	IF iCountRemote>=20 THEN //累计20s认为时间可用
		iCountRemote:=20;
		dDelRTime := TO_ULINT(stUTC_Timestamp) - (dRTime + 8 * 3600 *1000);
		GVL.bRemoteTimeLock:=TRUE;
		//对外部和本机时间差做1分钟的均值滤波
	END_IF
	//GVL.dRemoteTime:=stUTC_Timestamp*1000000 - dMeanDelRTime;
	dLastRTime:=dRTime;
	(*
	IF GVL.bRemoteTimeLock THEN
		dCountRemote:= dCountRemote + 1;
		IF dCountRemote < 10000 THEN
			dMeanDelRTime := (dMeanDelRTime*(dCountRemote-1) + dDelRTime)/dCountRemote;
		ELSE
			dCountRemote := 10000;
			dMeanDelRTime := (dMeanDelRTime*(dCountRemote-1) + dDelRTime)/dCountRemote; 	
			//iDiff:=ULINT_TO_DINT(Gvl.dPTPCSTTime-dLastCSTtime);
			//dLastCSTtime:=dCSTTime;
		END_IF
	END_IF
	*)
END_IF

ulACUTimeStamp := stUTC_Timestamp - dDelRTime;

END_PROGRAM

// Device/Application/GPRMC_1_1
PROGRAM GPRMC_1_1
VAR
        com_init:gcan.FB_Com_Init;                      //gcan.FB_Com_Init为串口初始化功能块，可设定串口端口号，串口波特率等参数
        com_read:gcan.FB_Com_Read ;                                //gcan.FB_Com_Read为串口接收功能块，用于通过接收串口发送给PLC的数据
        com_write:gcan.FB_Com_Write ;                        //gcan.FB_Com_Write为串口发送功能块，用于发送串口数据
        m_uiError:UINT;                                                        //用于承接功能块中报错引脚错误信息的变量
        m_out:BOOL;                                                                //用于承接功能块中完成标志引脚数据的变量
        isFirst:BOOL:=TRUE;                                                //用于判断初始化只执行一次的逻辑
        mPort:BYTE;                                                                //程序中用作设定串口端口号
        recSize:UINT;                                                        //接收数据长度，单位：字节
        recBuf:ARRAY[0..120] OF BYTE;                        //用于存放接收到的串口数据的数组
        iYear: INT;                             //年
        iMonth: INT;                            //月
        iDay: INT;                              //日
        iHour: INT;                             //时
        iMinute: INT;                           //分
        iSecond: INT;                           //秒
    bChecksumValid: BOOL := FALSE;                //校验和
        nFrameHeadPos: INT := 0;                //帧头索引          
    nPos        : INT;                      //帧头位置
    nChecksumRx : BYTE := 0;                //和校验
        strDateTimeNow : STRING;
        gnssTimestamp: ULINT;
        gnssTimestamplast:ULINT;
        icount:INT;
END_VAR

////////////////////////////////////////////////////////////////////////////////////////
//串口接收TOD报文解析
//日期：2025/05/15
//版本：V1.1
/////////////////////////////////////////////////////////////////////////////////////////

mPort:=1;                                                                //串口端口号设定，GCAN-PLC-400、GCAN-PLC-510、GCAN-PLC-511，1为232，2为485
                                                                                //GCAN-PLC-324、GCAN-PLC-326，1为第一路485，2为第2路485
IF isFirst THEN
        com_init(                                                        //串口初始化功能块
        EN_IN:=TRUE,                                                //串口初始化功能块使能
        xEnable:=TRUE,                                                //串口功能使能
        bPort:=mPort,                                                //串口端口号设定
        uiBaudrate:=115200,                                        //串口波特率设定
        bParity:=0,                                                        //串口奇偶校验设定，0为无校验，1为奇校验，2为偶检验
        bDatabits:=8,                                                //数据位设定
        bStopbits:=1,                                                //停止位设定
        EN_OUT=>m_out,                                                //串口初始化功能块执行完成标志位
        uiError=>m_uiError);                                //串口初始化功能块执行错误信息
        isfirst:=FALSE;                                                //执行一次初始化后关闭IF的条件使其之后进入ELSE程序段运行

ELSE
        
                com_read(                                                //串口读取功能块
                EN_in:=TRUE,                                        //读取功能块使能，为TRUE执行读取
                bPort:=mPort,                                        //串口端口号设定
                p_brxdata:=ADR(recBuf),                        //读取到的串口数据引脚为指针类型，使用ADR()指向自建数组将数据存放到数组中
                uiMaxsize:=240,                                        //设定最大读取长度
                EN_out=>m_out,                                        //串口读取功能块执行完成标志位******功能块执行完成不代表接收完成********
                uiRecSize=>recSize,                                //串口接收数据长度，单位：字节，大于0时说明接收到数据可用于判断是否接收
                uierror=>m_uierror);                        //串口读取功能块执行错误信息
                // 查找帧头 $X (36, 88)
                FOR nPos := 0 TO 119 DO
                        IF recBuf[nPos] = 36 AND recBuf[nPos + 1] = 88 THEN
                                nFrameHeadPos := nPos;
                                EXIT;
                        END_IF
                END_FOR
                //解析时间日期 
                IF nFrameHeadPos + 26 <= 120 THEN
                        iYear:=BYTE_TO_INT(recBuf[nFrameHeadPos+23]-48)*1000+BYTE_TO_INT(recBuf[nFrameHeadPos+24]-48)*100+BYTE_TO_INT(recBuf[nFrameHeadPos+25]-48)*10+BYTE_TO_INT(recBuf[26]-48);
                        iMonth:=BYTE_TO_INT(recBuf[nFrameHeadPos+20]-48)*10+BYTE_TO_INT(recBuf[nFrameHeadPos+21]-48);
                        iDay:=BYTE_TO_INT(recBuf[nFrameHeadPos+17]-48)*10+BYTE_TO_INT(recBuf[nFrameHeadPos+18]-48);
                        iHour:=BYTE_TO_INT(recBuf[nFrameHeadPos+7]-48)*10+BYTE_TO_INT(recBuf[nFrameHeadPos+8]-48)+8;
                        iMinute:=BYTE_TO_INT(recBuf[nFrameHeadPos+9]-48)*10+BYTE_TO_INT(recBuf[nFrameHeadPos+10]-48);
                        iSecond:=BYTE_TO_INT(recBuf[nFrameHeadPos+11]-48)*10+BYTE_TO_INT(recBuf[nFrameHeadPos+12]-48);
                        // 计算时间戳                
                        
                        strDateTimeNow := CONCAT(STR1 := 'DT#', STR2 := INT_TO_STRING(iYear));
                        strDateTimeNow := CONCAT(STR1 := strDateTimeNow, STR2 := '-');
                        strDateTimeNow := CONCAT(STR1 := strDateTimeNow, STR2 := INT_TO_STRING(iMonth));
                        strDateTimeNow := CONCAT(STR1 := strDateTimeNow, STR2 := '-');
                        strDateTimeNow := CONCAT(STR1 := strDateTimeNow, STR2 := INT_TO_STRING(iDay));
                        strDateTimeNow := CONCAT(STR1 := strDateTimeNow, STR2 := '-');
                        strDateTimeNow := CONCAT(STR1 := strDateTimeNow, STR2 := INT_TO_STRING(iHour));
                        strDateTimeNow := CONCAT(STR1 := strDateTimeNow, STR2 := ':');
                        strDateTimeNow := CONCAT(STR1 := strDateTimeNow, STR2 := INT_TO_STRING(iMinute));
                        strDateTimeNow := CONCAT(STR1 := strDateTimeNow, STR2 := ':');
                        strDateTimeNow := CONCAT(STR1 := strDateTimeNow, STR2 := INT_TO_STRING(iSecond));
                        
                        gnssTimestamplast:=gnssTimestamp;
                        gnssTimestamp := DT_TO_ULINT(TO_DT(strDateTimeNow)) * 1000;
                        GVL.stGNSS_Timestap := gnssTimestamp;                        
                END_IF
                
                IF gnssTimestamplast<>gnssTimestamp THEN
                        icount:=0;
                ELSE
                        icount:=icount+1;
                END_IF        
END_IF

END_PROGRAM

// Device/Application/PID_1
FUNCTION_BLOCK PID_1
VAR_INPUT
    rTarget : REAL;       (* 设定值 *)
    rFeedback : REAL;       (* 反馈值 *)
	rPosLimPositive:LREAL;//位置正限位
	rPosLimNegative:LREAL;//位置反限位
	rKp:REAL;     //比例增益
	rKi:REAL;     //积分增益
	rKd:REAL;     //微分增益
	iThreshold:INT;//积分项开启的位置阈值
	bPIDEnable:BOOL:=TRUE;//PID使能
	rVelLim:LREAL;//速度限制
END_VAR
VAR_OUTPUT
    rPIDOutput : LREAL:=0;         //带方向的输出速度

END_VAR
VAR
	//rPIDOutPut: REAL:=0.0;
	rLastError: LREAL:=0.0;(*上一次误差*)
	rErrorNow:LREAL:=0.0;(*当前误差*)
    rIntegralNew : LREAL := 0.0; (* 积分项 *)
    rDerivativeNew : LREAL := 0.0; (* 微分项 *)
	rDelta: LREAL;(*增量*)
	rProportionNew: LREAL;
	
	//iAzPIDEnable: INT;
END_VAR


IF (bPIDEnable>0) THEN //如果PID使能
	IF rTarget=rFeedback THEN
		rPIDOutput:=0;	
	ELSE
	
		rErrorNow:=rTarget-rFeedback;//计算当前误差 en
		rProportionNew:=rErrorNow;//比例项
		//积分项
		IF rFeedback>rPosLimNegative AND rFeedback<rPosLimPositive THEN //若在软限位之内，工作时开启积分项
			IF (ABS(rTarget-rFeedback)<iThreshold OR iThreshold = -1) THEN//位置差小于积分阈值开始积分，或者设置阈值为-1，不启用这个控制
				rIntegralNew:= rIntegralNew+rErrorNow; //积分项
			ELSE
				rIntegralNew:=0;
			END_IF;
		ELSE //不在软限位范围内,则积分项为0
			rIntegralNew:=0;
		END_IF

		//PID输出
		rPIDOutPut:=rKp*rProportionNew+rKi*rIntegralNew;


		//PID限速
		
			IF rPIDOutput<(-rVelLim) THEN
				rPIDOutput:=-rVelLim;
			ELSIF rPIDOutput>rVelLim THEN
				rPIDOutput:=rVelLim;
			END_IF
		
		
		IF rFeedback>rPosLimPositive AND rPIDOutput>0 THEN 
			rPIDOutput:=0;
		END_IF
		IF rFeedback<rPosLimNegative AND rPIDOutput<0 THEN
			rPIDOutput:=0;
		END_IF
		
		rLastError:=rErrorNow;//将当前误差赋值给上一次误差
		
	END_IF
ELSE//非使能清零PID各项
	rProportionNew:=0.0;
	rIntegralNew:=0.0;
	rPIDOutput:=0.0;
END_IF

END_FUNCTION_BLOCK

// Device/Application/PLC_PRG
PROGRAM PLC_PRG
VAR
	a : DINT;
	b : REAL;
END_VAR

a := REAL_TO_DINT(b * 524288 / 360);

END_PROGRAM

// Device/Application/XPTOD_SerialCom
PROGRAM XPTOD_SerialCom
VAR
        com_init:gcan.FB_Com_Init;                      //gcan.FB_Com_Init为串口初始化功能块，可设定串口端口号，串口波特率等参数
        com_read:gcan.FB_Com_Read ;                                //gcan.FB_Com_Read为串口接收功能块，用于通过接收串口发送给PLC的数据
        com_write:gcan.FB_Com_Write ;                        //gcan.FB_Com_Write为串口发送功能块，用于发送串口数据
        m_uiError:UINT;                                                        //用于承接功能块中报错引脚错误信息的变量
        m_out:BOOL;                                                                //用于承接功能块中完成标志引脚数据的变量
        isFirst:BOOL:=TRUE;                                                //用于判断初始化只执行一次的逻辑
        mPort:BYTE;                                                                //程序中用作设定串口端口号
        recSize:UINT;                                                        //接收数据长度，单位：字节
        recBuf:ARRAY[0..239] OF BYTE;                        //用于存放接收到的串口数据的数组
        iYear: INT;                             //年
        iMonth: INT;                            //月
        iDay: INT;                              //日
        iHour: INT;                             //时
        iMinute: INT;                           //分
        iSecond: INT;                           //秒
    bChecksumValid: BOOL := FALSE;                //校验和
        nFrameHeadPos: INT := 0;                //帧头索引          
    nPos        : INT;                      //帧头位置
    nChecksumRx : BYTE := 0;                //和校验
        strDateTimeNow : STRING;
        gnssTimestamp: ULINT;
        gnssTimestamplast:ULINT;
        icount:INT;
END_VAR

////////////////////////////////////////////////////////////////////////////////////////
//串口接收TOD报文解析
//日期：2025/05/15
//版本：V1.1
/////////////////////////////////////////////////////////////////////////////////////////

mPort:=1;                                                                //串口端口号设定，GCAN-PLC-400、GCAN-PLC-510、GCAN-PLC-511，1为232，2为485
                                                                                //GCAN-PLC-324、GCAN-PLC-326，1为第一路485，2为第2路485
IF isFirst THEN
        com_init(                                                        //串口初始化功能块
        EN_IN:=TRUE,                                                //串口初始化功能块使能
        xEnable:=TRUE,                                                //串口功能使能
        bPort:=mPort,                                                //串口端口号设定
        uiBaudrate:=115200,                                        //串口波特率设定
        bParity:=0,                                                        //串口奇偶校验设定，0为无校验，1为奇校验，2为偶检验
        bDatabits:=8,                                                //数据位设定
        bStopbits:=1,                                                //停止位设定
        EN_OUT=>m_out,                                                //串口初始化功能块执行完成标志位
        uiError=>m_uiError);                                //串口初始化功能块执行错误信息
        isfirst:=FALSE;                                                //执行一次初始化后关闭IF的条件使其之后进入ELSE程序段运行

ELSE
        
                com_read(                                                //串口读取功能块
                EN_in:=TRUE,                                        //读取功能块使能，为TRUE执行读取
                bPort:=mPort,                                        //串口端口号设定
                p_brxdata:=ADR(recBuf),                        //读取到的串口数据引脚为指针类型，使用ADR()指向自建数组将数据存放到数组中
                uiMaxsize:=240,                                        //设定最大读取长度
                EN_out=>m_out,                                        //串口读取功能块执行完成标志位******功能块执行完成不代表接收完成********
                uiRecSize=>recSize,                                //串口接收数据长度，单位：字节，大于0时说明接收到数据可用于判断是否接收
                uierror=>m_uierror);                        //串口读取功能块执行错误信息
                // 查找帧头 $X (36, 88)
                FOR nPos := 1 TO 240 DO
                        IF recBuf[nPos] = 36 AND recBuf[nPos + 1] = 88 THEN
                                nFrameHeadPos := nPos;
                                EXIT;
                        END_IF
                END_FOR
                //解析时间日期 
                IF nFrameHeadPos + 26 <= 240 THEN
                        iYear:=BYTE_TO_INT(recBuf[nFrameHeadPos+23]-48)*1000+BYTE_TO_INT(recBuf[nFrameHeadPos+24]-48)*100+BYTE_TO_INT(recBuf[nFrameHeadPos+25]-48)*10+BYTE_TO_INT(recBuf[26]-48);
                        iMonth:=BYTE_TO_INT(recBuf[nFrameHeadPos+20]-48)*10+BYTE_TO_INT(recBuf[nFrameHeadPos+21]-48);
                        iDay:=BYTE_TO_INT(recBuf[nFrameHeadPos+17]-48)*10+BYTE_TO_INT(recBuf[nFrameHeadPos+18]-48);
                        iHour:=BYTE_TO_INT(recBuf[nFrameHeadPos+7]-48)*10+BYTE_TO_INT(recBuf[nFrameHeadPos+8]-48)+8;
                        iMinute:=BYTE_TO_INT(recBuf[nFrameHeadPos+9]-48)*10+BYTE_TO_INT(recBuf[nFrameHeadPos+10]-48);
                        iSecond:=BYTE_TO_INT(recBuf[nFrameHeadPos+11]-48)*10+BYTE_TO_INT(recBuf[nFrameHeadPos+12]-48);
                        // 计算时间戳                
                        
                        strDateTimeNow := CONCAT(STR1 := 'DT#', STR2 := INT_TO_STRING(iYear));
                        strDateTimeNow := CONCAT(STR1 := strDateTimeNow, STR2 := '-');
                        strDateTimeNow := CONCAT(STR1 := strDateTimeNow, STR2 := INT_TO_STRING(iMonth));
                        strDateTimeNow := CONCAT(STR1 := strDateTimeNow, STR2 := '-');
                        strDateTimeNow := CONCAT(STR1 := strDateTimeNow, STR2 := INT_TO_STRING(iDay));
                        strDateTimeNow := CONCAT(STR1 := strDateTimeNow, STR2 := '-');
                        strDateTimeNow := CONCAT(STR1 := strDateTimeNow, STR2 := INT_TO_STRING(iHour));
                        strDateTimeNow := CONCAT(STR1 := strDateTimeNow, STR2 := ':');
                        strDateTimeNow := CONCAT(STR1 := strDateTimeNow, STR2 := INT_TO_STRING(iMinute));
                        strDateTimeNow := CONCAT(STR1 := strDateTimeNow, STR2 := ':');
                        strDateTimeNow := CONCAT(STR1 := strDateTimeNow, STR2 := INT_TO_STRING(iSecond));
                        
                        gnssTimestamplast:=gnssTimestamp;
                        gnssTimestamp := DT_TO_ULINT(TO_DT(strDateTimeNow)) * 1000;
                        GVL.stGNSS_Timestap := gnssTimestamp;                        
                END_IF
                
                IF gnssTimestamplast<>gnssTimestamp THEN
                        icount:=0;
                ELSE
                        icount:=icount+1;
                END_IF        
END_IF

END_PROGRAM

// Device/Application/插值模块/InterDataProcess
FUNCTION_BLOCK InterDataProcess
VAR_INPUT
	ulRealTime: ULINT;//实际时间 单位纳秒
	//aOrbitTime: ARRAY [1..5] OF ULINT;//轨道时间数组
	Arr: ARRAY [1..5] OF ULINT:=[9,0,1,5,4]; // 创建一个包含5个整数的数组 轨道时间数组  起点 1970-01-01 0:00:00 单位纳秒
    
END_VAR
VAR_OUTPUT
	MaxVal, MinVal: ULINT;   // 定义最大值、最小值和循环计数器变量
    MaxIndex, MinIndex: INT; // 定义最大值和最小值的索引
	ulInterRealTime : ULINT;//插值使用的时间
END_VAR
VAR
	i,j: INT;
END_VAR

//该功能块查找到轨道时间数组内最大最小值以及索引位置
//找出最大最小值
MaxVal := 0; // 初始化最大值
MinVal := 0; // 初始化最小值
MaxIndex := 0; // 初始化最大值的索引
MinIndex := 0; // 初始化最小值的索引

FOR i := 1 TO 5 DO
    IF Arr[i] <> 0 THEN
        IF MaxVal = 0 THEN
            MaxVal := Arr[i];
            MaxIndex := i;
        ELSIF Arr[i] > MaxVal THEN
            MaxVal := Arr[i];
            MaxIndex := i;
        END_IF

        IF MinVal = 0 THEN
            MinVal := Arr[i];
            MinIndex := i;
        ELSIF Arr[i] < MinVal THEN
            MinVal := Arr[i];
            MinIndex := i;
        END_IF
    END_IF
END_FOR

// MaxVal 和 MinVal 包含了最大值和最小值，不考虑值为0的元素
// MaxIndex 和 MinIndex 包含了最大值和最小值的索引


//当前时间和最大最小比较 
IF ulRealTime<MinVal*1000000 THEN //小于插值范围 取最小时间
	//
	ulInterRealTime:=MinVal*1000000; //应该修改插值位置 而不是时间
ELSIF ulRealTime>MaxVal*1000000THEN //大于插值范围 取最大时间
	//
	ulInterRealTime:=MaxVal*1000000;//应该修改插值位置 而不是时间
ELSE
	//如果内部有0 则不插值选取最新的数据
	FOR j:=1 TO 5 DO
		IF (Arr[i]=0) AND (j<5) THEN
			ulInterRealTime:=Arr[5];//应该修改插值位置 而不是时间
			MaxIndex:=5;
			EXIT;
		ELSIF (Arr[i]=0) AND (j=5) THEN
			//没有输入数据 需要报错吗？
		END_IF
	END_FOR
	//
END_IF

END_FUNCTION_BLOCK

// Device/Application/插值模块/LinearInter
FUNCTION_BLOCK LinearInter
VAR_INPUT
	tLastTime:ULINT;//上一时间
	rLastPos:REAL;//上一时间位置
	
	tCurTime:ULINT;//当前时间
	rCurPos:REAL;//当前时间位置
	
	tTargetTime:ULINT;//目标时间
END_VAR
VAR_OUTPUT
	rTargetpos:REAL;//目标时间位置
END_VAR
VAR
	iDelCurLastTime:LREAL:=1.0;//	当前与上一个时间差
	iDelTarCurTime:LREAL:=1.0;//目标与当前时间差
	rK:REAL;//方位斜率
END_VAR

//tLastTime:=tLastTime/1000000;
//tCurTime:=tCurTime/1000000;
//tTargetTime:=tTargetTime/1000000;
iDelTarCurTime:=ULINT_TO_LREAL(tTargetTime)-ULINT_TO_LREAL(tCurTime); //x1-x
IF (tCurTime-tLastTime)<>0 THEN
	iDelCurLastTime:=ULINT_TO_LREAL(tCurTime)-ULINT_TO_LREAL(tLastTime);  //x-x0
ELSE
	iDelCurLastTime:=1.0;
END_IF

IF iDelTarCurTime<>0 THEN
	rK:=(rCurPos-rLastPos)/(iDelCurLastTime);
ELSE
	rK:=0;
END_IF
rTargetpos:=rCurPos+rK*iDelTarCurTime;  //y1 + ((y1-y0)/(x1-x0))*(x-x1)

END_FUNCTION_BLOCK

// Device/Application/插值模块/threesimple2
FUNCTION_BLOCK threesimple2
VAR_INPUT
	aUTC_TIME:ARRAY [1..5] OF ULINT;  //用于三次样条插值的数据
	aPosCmd :ARRAY [1..5] OF LREAL;//用于三次样条插值的数据
	
	y0:REAL;
	yn:REAL;//y0,yn表示的是S''(x0)=f''(x0)=y0，S''(xn)=f''(xn)=yn,自然边界即条件值为0
	xt:REAL;//所求目标位置
END_VAR
VAR_OUTPUT
	sout:REAL;
	nout:INT;
END_VAR
VAR
	Three:three2;
	X:ARRAY [1..5] OF LREAL;
	Y:ARRAY [1..5] OF LREAL;
	M :ARRAY [1..5] OF LREAL;
	A: ARRAY [1..5,1..5] OF LREAL;
	D: ARRAY[1..3,1..3] OF LREAL;
	g: ARRAY [1..3] OF LREAL;
	h:ARRAY [1..4] OF LREAL;
	
	n:INT:=5;
	
	p1: ARRAY [1..4] OF REAL;
	p2:ARRAY [1..4] OF REAL;
	p3:ARRAY [1..4] OF REAL;
	p4:ARRAY [1..4] OF REAL;
	i:INT;
	
END_VAR

FOR i:=1 TO 5 DO
	X[i]:=ULINT_TO_LREAL(aUTC_TIME[i]);
	Y[i]:=aPosCmd[i];
END_FOR


Three(X:=X,Y:=Y,y0:=y0,yn:=yn,D=>D,h=>h,A=>A,g=>g,M=>M);

FOR i:=1 TO (n-1) DO
	p1[i]:=M[i]*(X[i+1]-xt)*(X[i+1]-xt)*(X[i+1]-xt)/(6*h[i]);
	p2[i]:=M[i+1]*(xt-X[i])*(xt-X[i])*(xt-X[i])/(6*h[i]);
	p3[i]:=(A[i,1]-M[i]/6*(h[i])*(h[i]))*(X[i+1]-xt)/h[i];
	p4[i]:=(A[i+1,1]-M[i+1]/6*(h[i])*(h[i]))*(xt-X[i])/h[i];
	
	
END_FOR


FOR i:=1 TO (n-1) DO
	IF (xt<=X[i+1])AND (xt>=X[i]) THEN
		nout:=i;
		sout:=p1[nout]+p2[nout]+p3[nout]+p4[nout]; 
	ELSIF xt>X[5] THEN
		nout:=4;
	ELSIF xt<X[1]THEN
		nout:=1;
	END_IF
END_FOR


//要不要判断插值模块是否有效？
sout:=p1[nout]+p2[nout]+p3[nout]+p4[nout]; 
(*
IF xt>X[5] THEN
	nout:=4;
	sout:=p1[nout]+p2[nout]+p3[nout]+p4[nout]; 
ELSIF xt<X[1] THEN
	nout:=1;
	sout:=p1[nout]+p2[nout]+p3[nout]+p4[nout]; 
END_IF
*)

END_FUNCTION_BLOCK

// /ElCtrl
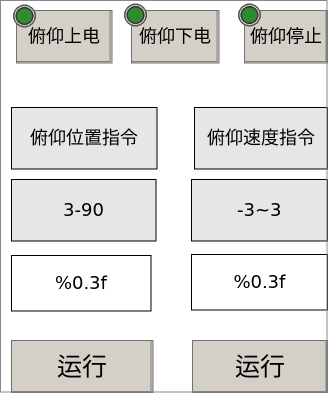
VISUALIZATION ElCtrl  // 328x393
    Button (131,10 88x53), "俯仰下电"
        OnMouseClick: execute { GVL.Axis1Local.iMode:=0; }
    Button (16,10 96x53), "俯仰上电"
        OnMouseClick: execute { GVL.Axis1Local.iMode:=1; }
    Lamp1 (6,3 37x26), variable: GVL.Axis1Status.bServo_Enable, style: Lamp-Lamp1-Green
    Lamp1 (117,2 37x26), variable: NOT(GVL.Axis1Status.bServo_Enable), style: Lamp-Lamp1-Green
    Button (244,10 84x53), "俯仰停止"
        OnMouseClick: execute { GVL.Axis1Local.iMode:=7; }
    Lamp1 (231,2 37x26), variable: NOT(GVL.Axis1Status.Moving), style: Lamp-Lamp1-Green
    Rectangle (11,107 146x62), "俯仰位置指令"
    Rectangle (11,255 140x56), "%0.3f", text variable: ElV.rPosCmd
        OnMouseClick: write the text variable via Default, min 3, max 90
    Button (11,340 142x53), "运行"
        OnMouseClick: execute {
            GVL.Axis1Local.rPosCmd:=GVL.ElV.rPosCmd+90;
            GVL.Axis1Local.iMode:=4;
            GVL.Axis1Local.bPIDEnable:=TRUE;
        }
    Rectangle (194,107 134x62), "俯仰速度指令"
    Rectangle (191,254 137x56), "%0.3f", text variable: ElV.rVelCmd
        OnMouseClick: write the text variable via Default, min -10, max 10
    Button (192,340 136x53), "运行"
        OnMouseClick: execute { GVL.Axis1Local.rVelCmd:=GVL.ElV.rVelCmd; GVL.Axis1Local.iMode:=3; }
    Rectangle (11,179 145x62), "3-90"
    Rectangle (191,179 137x62), "-3~3"
END_VISUALIZATION

// Device/Application/可视化/AzCtrl
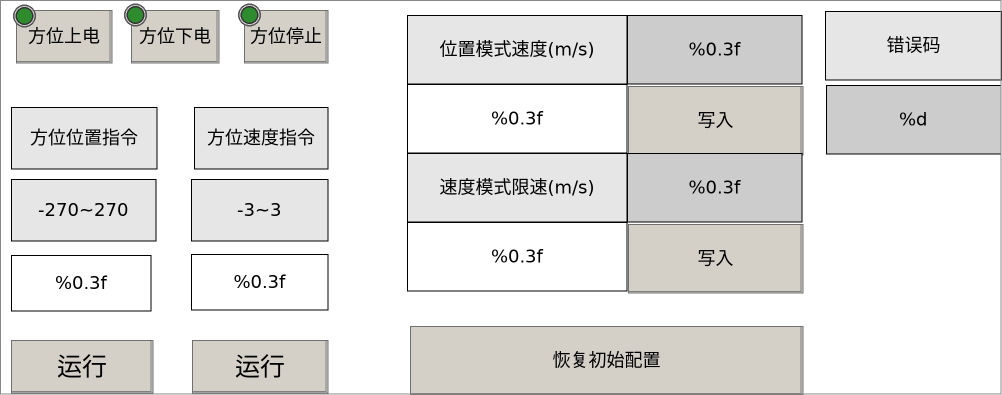
VISUALIZATION AzCtrl  // 1002x395
    Button (131,10 88x53), "方位下电"
        OnMouseClick: execute { GVL.Axis2Local.iMode:=0; }
    Button (16,10 96x53), "方位上电"
        OnMouseClick: execute { GVL.Axis2Local.iMode:=1; }
    Lamp1 (6,3 37x26), variable: GVL.Axis2Status.bServo_Enable, style: Lamp-Lamp1-Green
    Lamp1 (117,2 37x26), variable: NOT(GVL.Axis2Status.bServo_Enable), style: Lamp-Lamp1-Green
    Button (244,10 84x53), "方位停止"
        OnMouseClick: execute { GVL.Axis2Local.iMode:=7; }
    Lamp1 (231,2 37x26), variable: NOT(GVL.Axis2Status.Moving), style: Lamp-Lamp1-Green
    Rectangle (11,107 146x62), "方位位置指令"
    Rectangle (11,255 140x56), "%0.3f", text variable: AzV.rPosCmd
        OnMouseClick: write the text variable via Default, min -270, max 270
    Button (11,340 142x53), "运行"
        OnMouseClick: execute {
            GVL.Axis2Local.rPosCmd:=-GVL.AzV.rPosCmd;
            GVL.Axis2Local.iMode:=4;
            GVL.Axis2Local.bPIDEnable:=TRUE;
        }
    Rectangle (194,107 134x62), "方位速度指令"
    Rectangle (191,254 137x56), "%0.3f", text variable: AzV.rVelCmd
        OnMouseClick: write the text variable via Default, min -20, max 20
    Button (192,340 136x53), "运行"
        OnMouseClick: execute { GVL.Axis2Local.rVelCmd:=GVL.AzV.rVelCmd*(-1); GVL.Axis2Local.iMode:=3; }
    Rectangle (11,179 145x62), "-270~270"
    Rectangle (191,179 137x62), "-3~3"
    Rectangle (627,15 175x69), "%0.3f", text variable: Axis2Local.Pos_Vel
    Rectangle (407,15 220x69), "位置模式速度(m/s)"
    Rectangle (407,84 220x69), "%0.3f", text variable: AzV.Pos_Vel
        OnMouseClick: write the text variable via Edit, min -15.5, max 15.5
    Button (628,86 175x69), "写入"
        OnMouseClick: execute { Axis2Local.Pos_Vel:=AzV.Pos_Vel; }
    Rectangle (627,153 175x69), "%0.3f", text variable: Axis2Local.rVel_Limit
    Rectangle (407,153 220x69), "速度模式限速(m/s)"
    Rectangle (407,222 220x69), "%0.3f", text variable: AzV.rVel_Limit
        OnMouseClick: write the text variable via Edit, min 2, max 15.5
    Button (628,224 175x69), "写入"
        OnMouseClick: execute { Axis2Local.rVel_Limit:=AzV.rVel_Limit; }
    Button (410,326 393x69), "恢复初始配置"
        OnMouseClick: execute { Axis2Local.rVel_Limit:=3; Axis2Local.Pos_Vel:=4; }
    Rectangle (826,85 175x69), "%d", text variable: GVL.eAzErrorcode
    Rectangle (825,11 177x69), "错误码"
END_VISUALIZATION

// Device/Application/可视化/ElCtrl
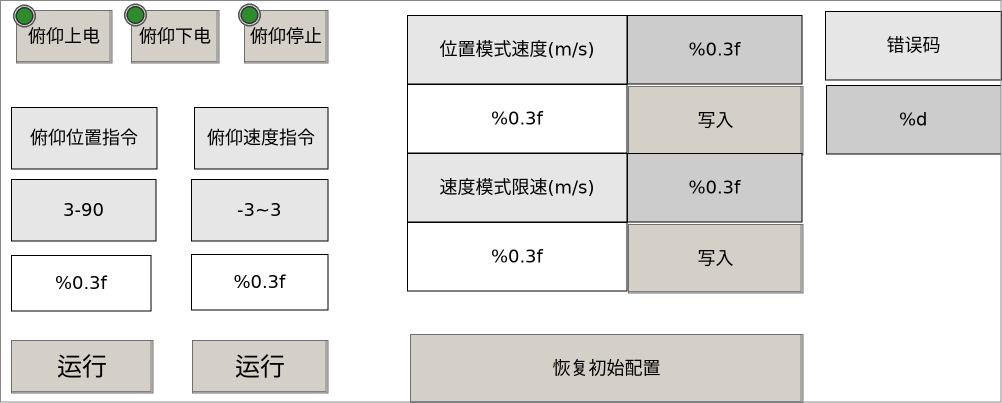
VISUALIZATION ElCtrl  // 1002x403
    Button (131,10 88x53), "俯仰下电"
        OnMouseClick: execute { GVL.Axis1Local.iMode:=0; }
    Button (16,10 96x53), "俯仰上电"
        OnMouseClick: execute { GVL.Axis1Local.iMode:=1; }
    Lamp1 (6,3 37x26), variable: GVL.Axis1Status.bServo_Enable, style: Lamp-Lamp1-Green
    Lamp1 (117,2 37x26), variable: NOT(GVL.Axis1Status.bServo_Enable), style: Lamp-Lamp1-Green
    Button (244,10 84x53), "俯仰停止"
        OnMouseClick: execute { GVL.Axis1Local.iMode:=7; }
    Lamp1 (231,2 37x26), variable: NOT(GVL.Axis1Status.Moving), style: Lamp-Lamp1-Green
    Rectangle (11,107 146x62), "俯仰位置指令"
    Rectangle (11,255 140x56), "%0.3f", text variable: ElV.rPosCmd
        OnMouseClick: write the text variable via Default, min 0, max 90
    Button (11,340 142x53), "运行"
        OnMouseClick: execute {
            GVL.Axis1Local.rPosCmd:=GVL.ElV.rPosCmd+90;
            GVL.Axis1Local.iMode:=4;
            GVL.Axis1Local.bPIDEnable:=TRUE;
        }
    Rectangle (194,107 134x62), "俯仰速度指令"
    Rectangle (191,254 137x56), "%0.3f", text variable: ElV.rVelCmd
        OnMouseClick: write the text variable via Default, min -13, max 13
    Button (192,340 136x53), "运行"
        OnMouseClick: execute { GVL.Axis1Local.rVelCmd:=GVL.ElV.rVelCmd; GVL.Axis1Local.iMode:=3; }
    Rectangle (11,179 145x62), "3-90"
    Rectangle (191,179 137x62), "-3~3"
    Rectangle (627,15 175x69), "%0.3f", text variable: Axis1Local.Pos_Vel
    Rectangle (407,15 220x69), "位置模式速度(m/s)"
    Rectangle (407,84 220x69), "%0.3f", text variable: ElV.Pos_Vel
        OnMouseClick: write the text variable via Edit, min -15.5, max 15.5
    Button (628,86 175x69), "写入"
        OnMouseClick: execute { Axis1Local.Pos_Vel:=ElV.Pos_Vel; }
    Rectangle (627,153 175x69), "%0.3f", text variable: Axis1Local.rVel_Limit
    Rectangle (407,153 220x69), "速度模式限速(m/s)"
    Rectangle (407,222 220x69), "%0.3f", text variable: ElV.rVel_Limit
        OnMouseClick: write the text variable via Edit, min 2, max 11
    Button (628,224 175x69), "写入"
        OnMouseClick: execute { Axis1Local.rVel_Limit:=ElV.rVel_Limit; }
    Button (410,334 393x69), "恢复初始配置"
        OnMouseClick: execute { Axis1Local.rVel_Limit:=3; Axis1Local.Pos_Vel:=4; }
    Rectangle (826,85 175x69), "%d", text variable: GVL.eElErrorcode
    Rectangle (825,11 177x69), "错误码"
END_VISUALIZATION

// Device/Application/可视化/north
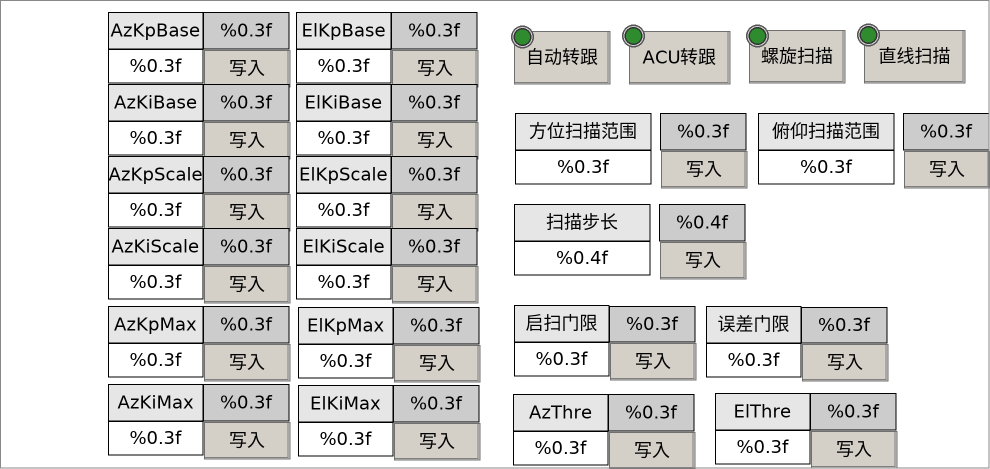
VISUALIZATION north  // 990x469
    Rectangle (203,12 86x37), "%0.3f", text variable: PersistentVars.rAzKpBase
    Rectangle (108,12 95x37), "AzKpBase"
    Rectangle (108,49 95x34), "%0.3f", text variable: GVL.rvAzKpBase
        OnMouseClick: write the text variable via Edit, min -100, max 100
    Button (204,50 86x37), "写入"
        OnMouseClick: execute { persistentvars.rAzKpBase := gvl.rvAzKpBase; }
    Rectangle (203,84 86x37), "%0.3f", text variable: PersistentVars.rAzKiBase
    Button (204,122 86x37), "写入"
        OnMouseClick: execute { persistentvars.rAzKiBase := gvl.rvAzKiBase; }
    Rectangle (203,156 86x37), "%0.3f", text variable: PersistentVars.rAzKpscale
    Button (204,194 86x37), "写入"
        OnMouseClick: execute { persistentvars.rAzKpScale := gvl.rvAzKpScale; }
    Rectangle (203,228 86x37), "%0.3f", text variable: PersistentVars.rAzKiscale
    Button (204,266 86x37), "写入"
        OnMouseClick: execute { persistentvars.rAzKiScale := gvl.rvAzKiScale; }
    Rectangle (108,84 95x37), "AzKiBase"
    Rectangle (108,121 95x34), "%0.3f", text variable: GVL.rvAzKiBase
        OnMouseClick: write the text variable via Edit, min -100, max 100
    Rectangle (108,156 95x37), "AzKpScale"
    Rectangle (108,193 95x34), "%0.3f", text variable: GVL.rvAzKpscale
        OnMouseClick: write the text variable via Edit, min -100, max 100
    Rectangle (108,228 95x37), "AzKiScale"
    Rectangle (108,265 95x34), "%0.3f", text variable: GVL.rvAzKiscale
        OnMouseClick: write the text variable via Edit, min -100, max 100
    Rectangle (391,12 86x37), "%0.3f", text variable: PersistentVars.rElKpBase
    Rectangle (296,12 95x37), "ElKpBase"
    Rectangle (296,49 95x34), "%0.3f", text variable: GVL.rvElKpBase
        OnMouseClick: write the text variable via Edit, min -100, max 100
    Button (392,50 86x37), "写入"
        OnMouseClick: execute { persistentvars.rElKpBase := gvl.rvElKpBase; }
    Rectangle (391,84 86x37), "%0.3f", text variable: PersistentVars.rElKiBase
    Button (392,122 86x37), "写入"
        OnMouseClick: execute { persistentvars.rElKiBase := gvl.rvElKiBase; }
    Rectangle (391,156 86x37), "%0.3f", text variable: PersistentVars.rElKpscale
    Button (392,194 86x37), "写入"
        OnMouseClick: execute { persistentvars.rElKpScale := gvl.rvElKpScale; }
    Rectangle (391,228 86x37), "%0.3f", text variable: PersistentVars.rElKiscale
    Button (392,266 86x37), "写入"
        OnMouseClick: execute { persistentvars.rElKiScale := gvl.rvElKiScale; }
    Rectangle (296,84 95x37), "ElKiBase"
    Rectangle (296,121 95x34), "%0.3f", text variable: GVL.rvElKiBase
        OnMouseClick: write the text variable via Edit, min -100, max 100
    Rectangle (296,156 95x37), "ElKpScale"
    Rectangle (296,193 95x34), "%0.3f", text variable: GVL.rvElKpscale
        OnMouseClick: write the text variable via Edit, min -100, max 100
    Rectangle (296,228 95x37), "ElKiScale"
    Rectangle (296,265 95x34), "%0.3f", text variable: GVL.rvElKiscale
        OnMouseClick: write the text variable via Edit, min -100, max 100
    Rectangle (203,306 86x37), "%0.3f", text variable: PersistentVars.rAzKpMax
    Rectangle (108,306 95x37), "AzKpMax"
    Rectangle (108,343 95x34), "%0.3f", text variable: GVL.rvAzKpMax
        OnMouseClick: write the text variable via Edit, min -100, max 100
    Button (204,344 86x37), "写入"
        OnMouseClick: execute { persistentvars.rAzKpMax := gvl.rvAzKpMax; }
    Rectangle (203,384 86x37), "%0.3f", text variable: PersistentVars.rAzKiMax
    Rectangle (108,384 95x37), "AzKiMax"
    Rectangle (108,421 95x34), "%0.3f", text variable: GVL.rvAzKiMax
        OnMouseClick: write the text variable via Edit, min -100, max 100
    Button (204,422 86x37), "写入"
        OnMouseClick: execute { persistentvars.rAzKiMax := gvl.rvAzKiMax; }
    Rectangle (393,307 86x37), "%0.3f", text variable: PersistentVars.rElKpMax
    Rectangle (298,307 95x37), "ElKpMax"
    Rectangle (298,344 95x34), "%0.3f", text variable: GVL.rvElKpMax
        OnMouseClick: write the text variable via Edit, min -100, max 100
    Button (394,345 86x37), "写入"
        OnMouseClick: execute { persistentvars.rElKpMax := gvl.rvElKpMax; }
    Rectangle (393,385 86x37), "%0.3f", text variable: PersistentVars.rElKiMax
    Rectangle (298,385 95x37), "ElKiMax"
    Rectangle (298,422 95x34), "%0.3f", text variable: GVL.rvElKiMax
        OnMouseClick: write the text variable via Edit, min -100, max 100
    Button (394,423 86x37), "写入"
        OnMouseClick: execute { persistentvars.rElKiMax := gvl.rvElKiMax; }
    Rectangle (608,394 86x37), "%0.3f", text variable: PersistentVars.rAzThre
    Rectangle (513,394 95x37), "AzThre"
    Rectangle (513,431 95x34), "%0.3f", text variable: GVL.rvAzThre
        OnMouseClick: write the text variable via Edit, min -100, max 100
    Button (609,432 86x37), "写入"
        OnMouseClick: execute { persistentvars.rAzThre := gvl.rvAzThre; }
    Rectangle (810,393 86x37), "%0.3f", text variable: PersistentVars.rElThre
    Rectangle (715,393 95x37), "ElThre"
    Rectangle (715,430 95x34), "%0.3f", text variable: GVL.rvElThre
        OnMouseClick: write the text variable via Edit, min -100, max 100
    Button (811,431 86x37), "写入"
        OnMouseClick: execute { persistentvars.rElThre := gvl.rvElThre; }
    Rectangle (609,306 86x36), "%0.3f", text variable: PersistentVars.rStartThre
    Rectangle (514,305 95x37), "启扫门限"
    Rectangle (514,342 95x34), "%0.3f", text variable: SecurityCheck.rSearchThreTemp
        OnMouseClick: write the text variable via Edit, min 0, max 5
    Button (610,343 86x37), "写入"
        OnMouseClick: execute { PersistentVars.rStartThre:=securitycheck.rSearchThreTemp; }
    Rectangle (660,113 86x37), "%0.3f", text variable: PersistentVars.rAzScanRange
    Rectangle (515,113 136x37), "方位扫描范围"
    Rectangle (515,150 136x34), "%0.3f", text variable: GVL.rAzScanRangeTemp
        OnMouseClick: write the text variable via Edit, min 0.1, max 1
    Button (661,151 86x37), "写入"
        OnMouseClick: execute { persistentvars.rAzScanRange := gvl.rAzScanRangeTemp; }
    Rectangle (903,113 86x37), "%0.3f", text variable: PersistentVars.rElScanRange
    Rectangle (758,113 136x37), "俯仰扫描范围"
    Rectangle (758,150 136x34), "%0.3f", text variable: GVL.rElScanRangeTemp
        OnMouseClick: write the text variable via Edit, min 0, max 1
    Button (904,151 86x37), "写入"
        OnMouseClick: execute { persistentvars.rElScanRange := gvl.rElScanRangeTemp; }
    Button (629,31 101x53), "ACU转跟"
        OnMouseClick: execute { PersistentVars.bTrackingMode:=FALSE; }
    Button (514,31 96x53), "自动转跟"
        OnMouseClick: execute { PersistentVars.bTrackingMode:=TRUE; }
    Lamp1 (504,24 37x26), variable: PersistentVars.bTrackingMode, style: Lamp-Lamp1-Green
    Lamp1 (615,23 37x26), variable: NOT(PersistentVars.bTrackingMode), style: Lamp-Lamp1-Green
    Button (864,30 101x53), "直线扫描"
        OnMouseClick: execute { PersistentVars.bSearchType:=FALSE; }
    Button (749,30 96x53), "螺旋扫描"
        OnMouseClick: execute { PersistentVars.bSearchType:=TRUE; }
    Lamp1 (739,23 37x26), variable: PersistentVars.bSearchType, style: Lamp-Lamp1-Green
    Lamp1 (850,22 37x26), variable: NOT(PersistentVars.bSearchType), style: Lamp-Lamp1-Green
    Rectangle (801,307 86x36), "%0.3f", text variable: PersistentVars.rErrorThre
    Rectangle (706,306 95x37), "误差门限"
    Rectangle (706,343 95x34), "%0.3f", text variable: GVL.rErrorTherTemp
        OnMouseClick: write the text variable via Edit, min 0, max 10
    Button (802,344 86x37), "写入"
        OnMouseClick: execute { PersistentVars.rErrorThre := GVL.rErrorTherTemp; }
    Rectangle (659,204 86x37), "%0.4f", text variable: PersistentVars.rStep
    Rectangle (514,204 136x37), "扫描步长"
    Rectangle (514,241 136x34), "%0.4f", text variable: GVL.rStepTemp
        OnMouseClick: write the text variable via Edit, min 0.0001, max 0.1
    Button (660,242 86x37), "写入"
        OnMouseClick: execute { persistentvars.rStep := gvl.rStepTemp; }
END_VISUALIZATION

// Device/Application/可视化/TlCtrl
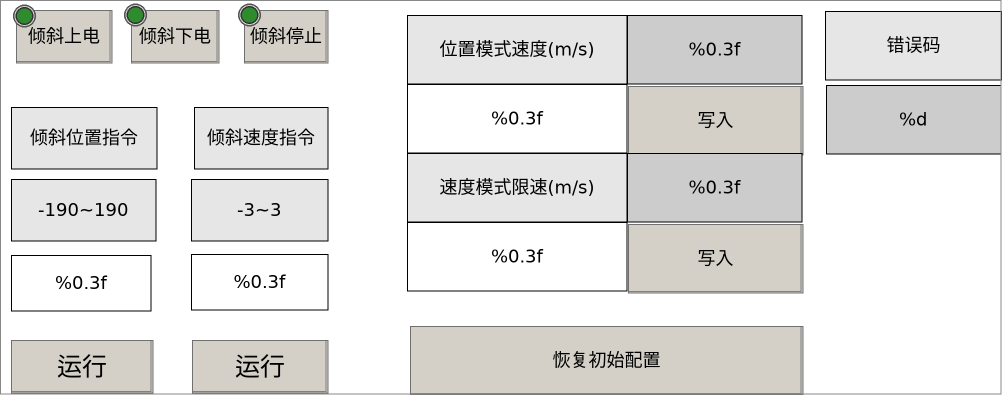
VISUALIZATION TlCtrl  // 1002x395
    Button (131,10 88x53), "倾斜下电"
        OnMouseClick: execute { GVL.Axis3Local.iMode:=0; }
    Button (16,10 96x53), "倾斜上电"
        OnMouseClick: execute { GVL.Axis3Local.iMode:=1; }
    Lamp1 (6,3 37x26), variable: GVL.Axis3Status.bServo_Enable, style: Lamp-Lamp1-Green
    Lamp1 (117,2 37x26), variable: NOT(GVL.Axis3Status.bServo_Enable), style: Lamp-Lamp1-Green
    Button (244,10 84x53), "倾斜停止"
        OnMouseClick: execute { GVL.Axis3Local.iMode:=7; }
    Lamp1 (231,2 37x26), variable: NOT(GVL.Axis3Status.Moving), style: Lamp-Lamp1-Green
    Rectangle (11,107 146x62), "倾斜位置指令"
    Rectangle (11,255 140x56), "%0.3f", text variable: TiV.rPosCmd
        OnMouseClick: write the text variable via Default, min -190, max 190
    Button (11,340 142x53), "运行"
        OnMouseClick: execute {
            GVL.Axis3Local.rPosCmd:=-GVL.TiV.rPosCmd;
            GVL.Axis3Local.iMode:=4;
            GVL.Axis3Local.bPIDEnable:=TRUE;
        }
    Rectangle (194,107 134x62), "倾斜速度指令"
    Rectangle (191,254 137x56), "%0.3f", text variable: TiV.rVelCmd
        OnMouseClick: write the text variable via Default, min -11, max 11
    Button (192,340 136x53), "运行"
        OnMouseClick: execute { GVL.Axis3Local.rVelCmd:=GVL.TiV.rVelCmd*(-1); GVL.Axis3Local.iMode:=3; }
    Rectangle (11,179 145x62), "-190~190"
    Rectangle (191,179 137x62), "-3~3"
    Rectangle (627,15 175x69), "%0.3f", text variable: Axis3Local.Pos_Vel
    Rectangle (407,15 220x69), "位置模式速度(m/s)"
    Rectangle (407,84 220x69), "%0.3f", text variable: TiV.Pos_Vel
        OnMouseClick: write the text variable via Edit, min -15.5, max 15.5
    Button (628,86 175x69), "写入"
        OnMouseClick: execute { Axis3Local.Pos_Vel:=TiV.Pos_Vel; }
    Rectangle (627,153 175x69), "%0.3f", text variable: Axis3Local.rVel_Limit
    Rectangle (407,153 220x69), "速度模式限速(m/s)"
    Rectangle (407,222 220x69), "%0.3f", text variable: TiV.rVel_Limit
        OnMouseClick: write the text variable via Edit, min -15.5, max 15.5
    Button (628,224 175x69), "写入"
        OnMouseClick: execute { Axis3Local.rVel_Limit:=TiV.rVel_Limit; }
    Button (410,326 393x69), "恢复初始配置"
        OnMouseClick: execute { Axis3Local.rVel_Limit:=3; Axis3Local.Pos_Vel:=4; }
    Rectangle (826,85 175x69), "%d", text variable: GVL.eTiErrorcode
    Rectangle (825,11 177x69), "错误码"
END_VISUALIZATION

// Device/Application/可视化/Visualization
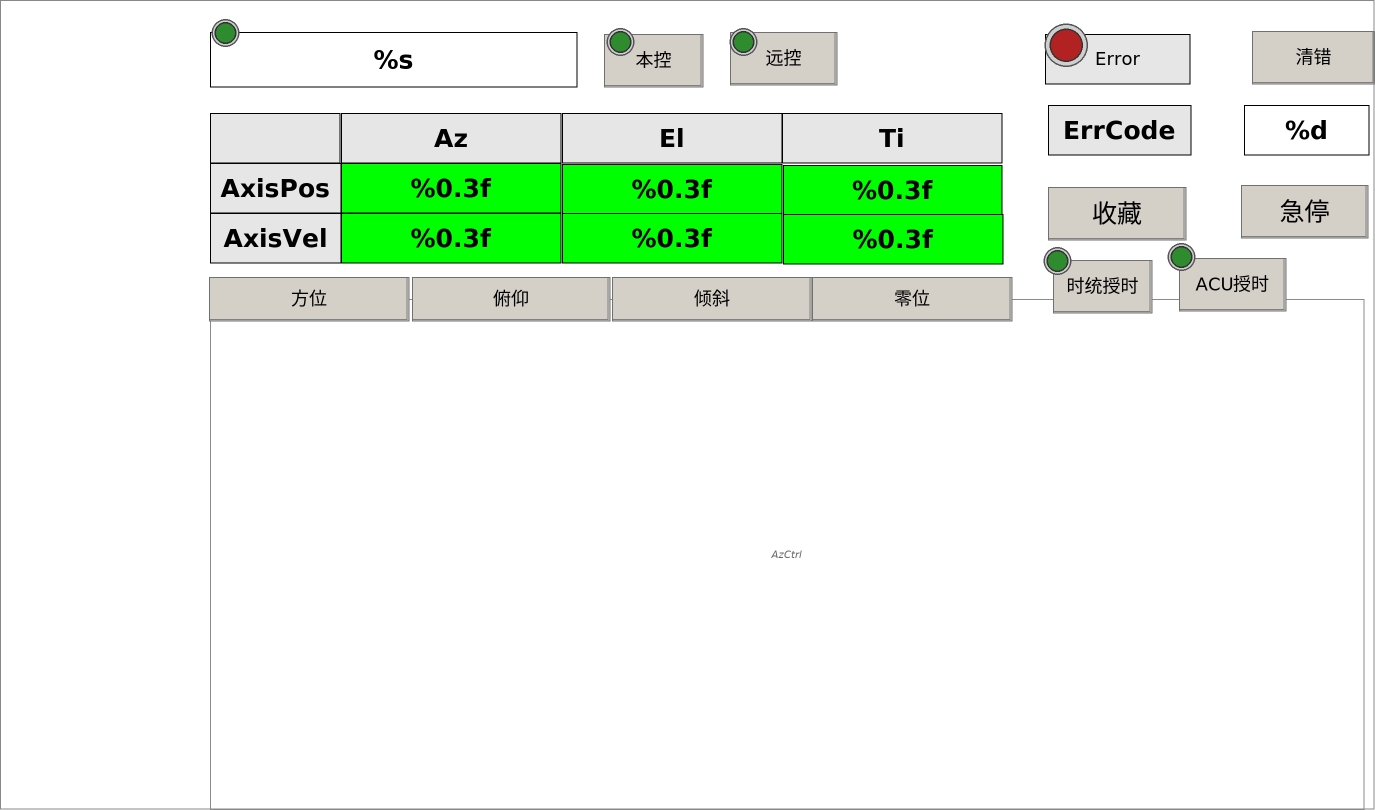
VISUALIZATION Visualization  // 1375x810
    Rectangle (210,32 367x55), "%s", text variable: RealTimePosCal.dtReal
    Button (604,34 99x53), "本控"
        OnMouseClick: execute { GVL.bLocalCtrl:=TRUE; }
    Button (730,32 107x53), "远控"
        OnMouseClick: execute { GVL.bLocalCtrl:=FALSE; }
    Lamp1 (596,26 49x32), variable: GVL.bLocalCtrl, style: Lamp-Lamp1-Green
    Lamp1 (721,26 45x32), variable: NOT(GVL.bLocalCtrl), style: Lamp-Lamp1-Green
    Rectangle (341,113 220x50), "Az"
    Rectangle (562,113 220x50), "El"
    Rectangle (210,163 131x50), "AxisPos"
    Rectangle (341,163 220x50), "%0.3f", text variable: GVL.rFctPosReal_2*(-1)
    Rectangle (562,164 220x50), "%0.3f", text variable: GVL.rFctPosReal_1-90
    Rectangle (210,113 130x50)
    Rectangle (210,213 131x50), "AxisVel"
    Rectangle (341,213 220x50), "%0.3f", text variable: GVL.rFctVelReal_2*(-1)
    Rectangle (562,213 220x50), "%0.3f", text variable: GVL.rFctVelReal_1
    Lamp1 (203,17 45x32), variable: TimeCase.Triger, style: Lamp-Lamp1-Green
    Rectangle (1045,34 145x50), "Error"
    Lamp1 (1026,20 80x50), variable: Az_ctrl_1.bVisError, style: Lamp-Lamp1-Red
    Button (1048,187 138x53), "收藏"
        OnMouseClick: execute {
            GVL.Axis1Local.rPosCmd:=180;
            GVL.Axis1Local.iMode:=4;
            GVL.Axis1Local.bPIDEnable:=TRUE;
            GVL.Axis2Local.rPosCmd:=0;
            GVL.Axis2Local.iMode:=4;
            GVL.Axis2Local.bPIDEnable:=TRUE;
            GVL.Axis3Local.rPosCmd:=0;
            GVL.Axis3Local.iMode:=4;
            GVL.Axis3Local.bPIDEnable:=TRUE;
        }
    Button (1241,185 127x53), "急停"
        OnMouseClick: execute {
            GVL.Axis1Local.iMode:=0;
            GVL.Axis2Local.iMode:=0;
            GVL.Axis3Local.iMode:=0;
        }
    Rectangle (1048,105 143x50), "ErrCode"
    Rectangle (1244,105 125x50), "%d", text variable: GVL.Error_code
    Button (1252,31 123x53), "清错"
        OnMouseClick: execute { GVL.bError_Reset:=TRUE; }
    Rectangle (782,113 220x50), "Ti"
    Rectangle (783,165 219x50), "%0.3f", text variable: GVL.rFctPosReal_3*(-1)
    Rectangle (783,214 220x50), "%0.3f", text variable: GVL.rFctVelReal_3*(-1)
    TabControl (210,299 1154x511), frame switch variable: GVL.iVisualSwitch
        shows AzCtrl()
        shows ElCtrl()
        shows TlCtrl()
        shows north()
        shows IOtest()
        shows IOState()
    Button (209,277 200x44), "方位", input disabled if: GVL.bAzVisable
        OnMouseClick: execute {
            GVL.bAzVisable:=TRUE;
            GVL.bElVisable:=FALSE;
            GVL.bTlVisable:=FALSE;
            GVL.bLocalAutoTrackVis:=FALSE;
            GVL.iVisualSwitch:=0;
        }
    Button (412,277 198x44), "俯仰", input disabled if: GVL.bElVisable
        OnMouseClick: execute {
            GVL.bAzVisable:=FALSE;
            GVL.bElVisable:=TRUE;
            GVL.bTlVisable:=FALSE;
            GVL.bLocalAutoTrackVis:=FALSE;
            GVL.iVisualSwitch:=1;
        }
    Button (612,277 200x44), "倾斜", input disabled if: GVL.bTlVisable
        OnMouseClick: execute {
            GVL.bAzVisable:=FALSE;
            GVL.bElVisable:=FALSE;
            GVL.bTlVisable:=TRUE;
            GVL.bLocalAutoTrackVis:=FALSE;
            GVL.iVisualSwitch:=2;
        }
    Button (812,277 200x44), "零位", input disabled if: GVL.bLocalAutoTrackVis
        OnMouseClick: execute {
            GVL.bAzVisable:=FALSE;
            GVL.bElVisable:=FALSE;
            GVL.bTlVisable:=FALSE;
            GVL.bLocalAutoTrackVis:=TRUE;
            GVL.iVisualSwitch:=3;
        }
    Button (1053,260 99x53), "时统授时"
        OnMouseClick: execute { GVL.bTimeSwich := FALSE; }
    Button (1179,258 107x53), "ACU授时"
        OnMouseClick: execute { GVL.bTimeSwich := TRUE; }
    Lamp1 (1033,245 49x32), variable: NOT(GVL.bTimeSwich), style: Lamp-Lamp1-Green
    Lamp1 (1159,241 45x32), variable: GVL.bTimeSwich, style: Lamp-Lamp1-Green
END_VISUALIZATION
